FUNCTION_BLOCK FB_StationMitZufUndVer EXTENDS FB_StationMitZuf
VAR_INPUT
	ifTeilBereitstellen:		IF_TeilBereitstellen;
END_VAR
VAR_OUTPUT
END_VAR
VAR
	eBereitstellStatus:		AblaufStatus := AblaufStatus.bereit;
	eStatusZuf:				StatusZufuehrung;
	
	nBereitstellZaehler:	INT;
	nAusschussZaehlerBerSt: INT;
END_VAR

//********************************************************************************					
//Schrittbetrieb
fbSchrittbetrieb.eBereitstellStatus := eBereitstellStatus;
fbSchrittbetrieb.bAblaufAktiv := nBereitstellZaehler > 0;

//********************************************************************************					
//Handzyklus (Muss Vor SUPER Call sein, damit diese Version vom Hand Zyklus ausgeführt wird)
//IF			bBtnHandZyklus THEN
//	bBtnHandZyklus := FALSE;
//	
//	IF			stStationInfo.bZyklusFertig
//		AND		bRstInPos
//		AND NOT MAIN.bProduzieren THEN
//		IF			MAIN.hatAufnBeiStJob(stStationInfo.nStationsNr) THEN							//Aufnahme will bearbeitet werden (Teile wurden schon bestellt)
//			ifStation.bearbeitenAnfordern(MAIN.getAufnahmeBeiStation(stStationInfo.nStationsNr));	//Aktuelle Aufnahme wird verwendet
//		ELSE																						//Aufnahme will NICHT bearbeitet werden (Teile müssen bestellt werden)
//			MAIN.vorwahlPseudoaufnahme();
//			ifTeilBereitstellen.holenAnfordern();
//			ifStation.bearbeitenAnfordern(Parameter.cAnzAufnahmen+1);								//Pseudoaufnahme wird verwendet
//		END_IF	
//	END_IF
//END_IF

//********************************************************************************					
//Call Basisklasse
SUPER^(stStationInfo := stStationInfo);

//********************************************************************************					
//Ablauf

IF			stStationInfo.bInitBeendet 
	AND NOT stStationInfo.bReset
	AND NOT fbSchrittbetrieb.bInQueue THEN
	
	IF			nBereitstellZaehler > 0 THEN
		ifTeilBereitstellen.teilBereitstellen();
	END_IF
END_IF

IF			(nAusschussZaehlerBerSt > 0)
	AND		(nBereitstellZaehler > 1
	OR		(nBereitstellZaehler > 0
	AND		(eBereitstellStatus = AblaufStatus.bereit))) THEN
	nBereitstellZaehler := nBereitstellZaehler-1;
	nAusschussZaehlerBerSt := nAusschussZaehlerBerSt-1;
END_IF

METHOD ausschussMelden
VAR_INPUT
END_VAR
SUPER^.ausschussMelden();
nAusschussZaehlerBerSt := nAusschussZaehlerBerSt+1;
END_METHOD

METHOD holenAnfordern
VAR_INPUT
END_VAR
nTeileZaehler := nTeileZaehler+1;
nBereitstellZaehler := nBereitstellZaehler+1;
END_METHOD

END_FUNCTION_BLOCK

(* stored: Version 1.1.0.1, ProductVersion 3.1.4024.12
   POU FB_StationMitZufUndVer: Id {a6cdbfaa-9822-4cdd-a675-e73e066f8662}, SpecialFunc None
   Method ausschussMelden: Id {9f2947bc-b965-406c-aea5-e687c63c0a28}
   Method holenAnfordern: Id {f412bbbf-339b-4746-bdff-41b4451e6782} *)
